PROGRAM pMsg
VAR
	msg: MsgPush;
END_VAR

METHOD PUBLIC Push_Alarm : BOOL
VAR_INPUT
	STR : WSTRING;
END_VAR
msg.iMessageId := 0;
msg.msgeLevel := MsgLevel.Alarm;
msg.sMessageStr1:=STR;
msg();
END_METHOD

METHOD PUBLIC Push_Alarm_NoPause : BOOL
VAR_INPUT
	STR : WSTRING;
END_VAR
msg.iMessageId := 0;
msg.msgeLevel := MsgLevel.Alarm;
msg.sMessageStr1:=STR;
msg();
END_METHOD

METHOD PUBLIC Push_Error : BOOL
VAR_INPUT
	STR : WSTRING;
END_VAR
msg.iMessageId := 0;
msg.msgeLevel := MsgLevel.Error;
msg.sMessageStr1:=STR;
SystemError := TRUE;
msg();
END_METHOD

METHOD PUBLIC Push_Info : BOOL
VAR_INPUT
	STR : WSTRING;
	
END_VAR
msg.iMessageId := 0;
msg.msgeLevel := MsgLevel.Info;
msg.sMessageStr1:=STR;
msg();
END_METHOD

END_PROGRAM

(* stored: Version 1.1.0.1, ProductVersion 3.1.4026.13
   POU pMsg: Id {7684ad6c-3919-4817-89f5-688b11f53eca}, SpecialFunc None
   Method Push_Alarm: Id {6bc02747-6728-4e1d-8f9b-d8d9f442df63}
   Method Push_Alarm_NoPause: Id {93c2844d-3181-4b3c-8a8e-46fab90054ba}
   Method Push_Error: Id {f3976628-e386-43b2-9ac6-20526979b396}
   Method Push_Info: Id {01d39928-1653-495f-8f78-34e7137ec7e7} *)
